FUNCTION_BLOCK FB_Figures
VAR_INPUT
END_VAR
VAR_OUTPUT
END_VAR
VAR
END_VAR

END_FUNCTION_BLOCK

(* stored: Version 1.1.0.1, ProductVersion 3.1.4024.12
   POU FB_Figures: Id {51316db0-3fb6-4d69-917d-1a96e95ae44e}, SpecialFunc None *)
